	FUNCTION_BLOCK FB 1015
	TITLE =A_2935_MXZ01MA BELT CONVEYOR 7400
	//COPYRIGHT:     (C) 2009  BUHLER AG, CH-9240 UZWIL, SWITZERLAND
	//
	//PRODUCT:       WinCoS_BIW01_09
	//
	//TITLE:         BELT CONVEYOR 7400
	//
	//--------------------------------------------------------------------------------
	//
	//IDENT:         AUTHOR:             DEPT:                             DATE:
	//
	//P01_FB1015.1.0 K.Renz              CSB41                             08.Jun.2010
	//               1st Release
	//
	//--------------------------------------------------------------------------------
	//
	//PURPOSE:
	//
	//MANUAL :
	//
	//RESTRICTIONS:
	//
	//--------------------------------------------------------------------------------
	AUTHOR  : KR
	FAMILY  : USW
	VERSION : 0.0


	VAR
	         Ma :  UDT 20500  ;  // Machine
	         Mon1  : FB14 ;    // spare
	         A_2935_SHE20 : FB14;  // Mon2: DigInpCont
	         A_2935_SHE21 : FB14;  // Mon3: DigInpCont
	         A_2935_BSA13 : FB14;  // Mon4: DigInpCont
	         A_2935_BZS14_15 : FB14;  // Mon5: DigInpCont
	         A_2935_BZS16_17 : FB14;   // Mon6: DigInpCont
	         A_2935_MXZ01 : FB12; // Motor: Motor
	END_VAR

	BEGIN
	NETWORK
	TITLE =Call SSW
	   UC  FB50
	END_FUNCTION_BLOCK
